{attribute 'linkalways'} 
{attribute 'no_explicit_call' := 'This FB is a CLASS and must be accessed using methods or properties'}
{attribute 'enable_dynamic_creation'}
FUNCTION_BLOCK Axis EXTENDS CyclicInstance
VAR
	_axisRef : Tc2_MC2.AXIS_REF;
	_power : MC_Power;
	_jog : MC_Jog;
	_readStatus : MC_ReadStatus;
	_parameterSet : ST_AxisParameterSet;
	
	_enable : BOOL;
	_enablePositive : BOOL;
	_enableNegative : BOOL;
	
	_override : LREAL := 100.0;
	_powerBufferMode : AxisBufferMode := AxisBufferMode.Aborting;
END_VAR

PROPERTY INTERNAL _InternalAxisRef : REFERENCE TO Tc2_MC2.AXIS_REF
GET
_InternalAxisRef REF= _axisRef;
END_GET
END_PROPERTY

PROPERTY INTERNAL _InternalJog : REFERENCE TO MC_Jog
GET
_InternalJog REF= _jog;
END_GET
END_PROPERTY

PROPERTY INTERNAL _InternalParameterSet : REFERENCE TO ST_AxisParameterSet
GET
_InternalParameterSet REF= _parameterSet;
END_GET
END_PROPERTY

PROPERTY AxisId : UDINT
GET
AxisId := _axisRef.NcToPlc.AxisId;
END_GET
END_PROPERTY

{warning 'add property implementation'}
PROPERTY BufferMode : Tc2_MC2.MC_BufferMode
GET
END_GET
SET
END_SET
END_PROPERTY

PROPERTY Busy : BOOL
GET
END_GET
END_PROPERTY

METHOD  CyclicCall
VAR_INST
	_readParameterSet : MC_ReadParameterSet;
	parameterSetRead : BOOL;
END_VAR
_power(
	Axis := THIS^._axisRef,
	Enable := THIS^._enable,
	Enable_Positive := THIS^._enablePositive,
	Enable_Negative := THIS^._enableNegative,
	Override := THIS^._override,
	BufferMode := THIS^._powerBufferMode
);

_readStatus(
	Axis := THIS^._axisRef,
	Enable := _enable
);

IF NOT parameterSetRead THEN
	_readParameterSet(
		Axis := THIS^._axisRef,
		Parameter := _parameterSet,
		Execute := TRUE
	);
	
	IF NOT _readParameterSet.Busy THEN
		_readParameterSet(
			Axis := THIS^._axisRef,
			Parameter := _parameterSet,
			Execute := TRUE
		);
		IF _readParameterSet.Done THEN
			parameterSetRead := TRUE;
		END_IF
	END_IF
END_IF
END_METHOD

METHOD Disable
_enable := FALSE;
END_METHOD

METHOD DisableNegative
_enableNegative := FALSE;
END_METHOD

METHOD DisablePositive
_enablePositive := FALSE;
END_METHOD

METHOD Enable
VAR_INPUT
	bufferMode : AxisBufferMode;
END_VAR
_enable := TRUE;
_powerBufferMode := bufferMode;
END_METHOD

METHOD EnableNegative : BOOL
_enableNegative := TRUE;
END_METHOD

METHOD EnablePositive
_enablePositive := TRUE;
END_METHOD

PROPERTY ErrorId : UDINT
GET
ErrorId := _readStatus.ErrorID;
END_GET
END_PROPERTY

METHOD Halt
VAR_INPUT
	feedback : REFERENCE TO I_CommandFeedback;
END_VAR
VAR_INST
	pCmd : POINTER TO HaltCommand;
END_VAR
pCmd := __NEW(HaltCommand(axisRef := THIS^));
pCmd^.Execute(feedback).ThenRelease();
END_METHOD

PROPERTY HasError : BOOL
GET
HasError := _readStatus.Error;
END_GET
END_PROPERTY

METHOD HomingBuilder : I_HomingBuilder
VAR_INST
	builder : DefaultHomingBuilder(axisRef := THIS^);
END_VAR
HomingBuilder := builder;
END_METHOD

PROPERTY IsAccelerating : BOOL
GET
IsAccelerating := _readStatus.Accelerating;
END_GET
END_PROPERTY

PROPERTY IsAtConstantVelocity : BOOL
GET
IsAtConstantVelocity := _readStatus.ConstantVelocity;
END_GET
END_PROPERTY

PROPERTY IsAtStandStill : BOOL
GET
IsAtStandStill := _readStatus.StandStill;
END_GET
END_PROPERTY

PROPERTY IsDecelerating : BOOL
GET
IsDecelerating := _readStatus.Decelerating;
END_GET
END_PROPERTY

PROPERTY IsErrorStopped : BOOL
GET
IsErrorStopped := _readStatus.ErrorStop;
END_GET
END_PROPERTY

PROPERTY IsHoming : BOOL
GET
IsHoming := _readStatus.Homing;
END_GET
END_PROPERTY

PROPERTY IsInContinuousMotion : BOOL
GET
IsInContinuousMotion := _readStatus.ContinuousMotion;
END_GET
END_PROPERTY

PROPERTY IsInDiscreteMotion : BOOL
GET
IsInDiscreteMotion := _readStatus.DiscreteMotion;
END_GET
END_PROPERTY

PROPERTY IsInSynchronizedMotion : BOOL
GET
IsInSynchronizedMotion := _readStatus.SynchronizedMotion;
END_GET
END_PROPERTY

PROPERTY IsReady : BOOL
GET
IsReady := _power.Status;
END_GET
END_PROPERTY

PROPERTY IsStatusValid : BOOL
GET
IsStatusValid := _readStatus.Valid;
END_GET
END_PROPERTY

PROPERTY IsStopping : BOOL
GET
IsStopping := _readStatus.Stopping;
END_GET
END_PROPERTY

METHOD JogBackwards
VAR_INPUT
	velocity : LREAL;
END_VAR
_jog(
	Axis := _axisRef,
	JogForward := FALSE,
	JogBackwards := TRUE,
	Mode := MC_JOGMODE_CONTINOUS,
	Velocity := velocity
);
END_METHOD

METHOD JogForward
VAR_INPUT
	velocity : LREAL;
END_VAR
_jog(
	Axis := _axisRef,
	JogForward := TRUE,
	JogBackwards := FALSE,
	Mode := MC_JOGMODE_CONTINOUS,
	Velocity := velocity
);
END_METHOD

METHOD MoveBuilder : I_MoveBuilder
VAR_INST
	builder : DefaultMoveBuilder(axisRef := THIS^);
END_VAR
MoveBuilder := builder;
END_METHOD

PROPERTY Override : LREAL
GET
Override := _override;
END_GET
SET
_override := Override;
END_SET
END_PROPERTY

METHOD Reset
VAR_INPUT
	feedback : REFERENCE TO I_CommandFeedback;
END_VAR
VAR_INST
	pCmd : POINTER TO ResetCommand;
END_VAR
pCmd := __NEW(ResetCommand(axisRef := THIS^));
pCmd^.Execute(feedback).ThenRelease();
END_METHOD

METHOD SetPositionAbsolute
VAR_INPUT
	positionToSet : LREAL;
	feedback : REFERENCE TO I_CommandFeedback;
END_VAR
VAR_INST
	pCmd : POINTER TO SetPositionCommand;
END_VAR
pCmd := __NEW(SetPositionCommand(axisRef := THIS^, position := positionToSet, mode := SetPositionMode.Absolute));
pCmd^.Execute(feedback).ThenRelease();
END_METHOD

METHOD SetPositionRelative
VAR_INPUT
	distanceToShift : LREAL;
	feedback : REFERENCE TO I_CommandFeedback;
END_VAR
VAR_INST
	pCmd : POINTER TO SetPositionCommand;
END_VAR
pCmd := __NEW(SetPositionCommand(axisRef := THIS^, position := distanceToShift, mode := SetPositionMode.Relative));
pCmd^.Execute(feedback).ThenRelease();
END_METHOD

METHOD Stop
VAR_INPUT
	feedback : REFERENCE TO I_CommandFeedback;
END_VAR
VAR_INST
	pCmd : POINTER TO StopCommand;
END_VAR
pCmd := __NEW(StopCommand(axisRef := THIS^));
pCmd^.Execute(feedback).ThenRelease();
END_METHOD

METHOD StopJogging
_jog(
	Axis := _axisRef,
	JogForward := FALSE,
	JogBackwards := FALSE,
);
END_METHOD

END_FUNCTION_BLOCK

(* stored: Version 1.1.0.1, ProductVersion 3.1.4024.12
   POU Axis: Id {2aaf2d97-dcbd-4e4f-bb30-8168c2228304}, SpecialFunc None
   Folder Actions: Id {d3a6f6e5-0dc6-41bb-8fed-2d69291737e9}
   Folder Builders: Id {8b93d50b-0153-46ae-83ea-c4e3e102f098}
   Folder Internal Methods: Id {a404c9ad-82b3-4270-92e5-46406a4ee946}
   Folder Internal Properties: Id {ff3545d4-cf9d-4f1c-9c6a-4608c8343033}
   Folder Properties: Id {bcfa7b74-d450-4ebb-b173-8da30bff7c11}
   Property _InternalAxisRef: Id {90609a99-e5bd-4b83-a58a-33c30ccc26cb}
   Get Get: Id {3b2ee038-497c-4033-a9b8-e83a2391191c}
   Property _InternalJog: Id {81758ae0-123d-466a-a4f8-f7ea636e9aab}
   Get Get: Id {8cd6a88b-f9db-4297-8b57-8b361f25d990}
   Property _InternalParameterSet: Id {247c45f2-47fd-4c00-8a9c-f77b32401e79}
   Get Get: Id {e12d2eff-e487-46f7-9fd3-f34e9951cc7f}
   Property AxisId: Id {67de2fd0-4aba-0578-2c2c-7b4e6a0d9ac8}
   Get Get: Id {821606fd-2277-088b-2511-fa15594f6c0e}
   Property BufferMode: Id {d3f9ce10-8ed2-4c86-bbbf-2cd31077c031}
   Get Get: Id {cb7a3b58-9630-4fcc-a8b2-6febff3711f9}
   Set Set: Id {90ad7435-fc63-4033-8f56-5ec9006dd1f3}
   Property Busy: Id {c365381d-4981-4e80-ad93-d15d1877f546}
   Get Get: Id {bb4c1cbb-227d-474b-b0fd-1dc32af91f9d}
   Method CyclicCall: Id {d18012b0-9520-4a5f-86ea-978a26c54f8e}
   Method Disable: Id {17b30872-fcd4-488a-b1b6-7fa79c000037}
   Method DisableNegative: Id {09f6abf1-b00f-4bfb-88e9-6ee7e9ba6e8f}
   Method DisablePositive: Id {59728fb8-b0dd-4aa9-bc80-abeb26875c9a}
   Method Enable: Id {c9911178-c912-485d-91e6-84927ecfc191}
   Method EnableNegative: Id {4800b13a-5042-4e28-861b-962c18550409}
   Method EnablePositive: Id {f7745032-8e58-4ba9-a609-48f560d8e17f}
   Property ErrorId: Id {ca7b6c5d-7148-4955-9c48-485f289f249e}
   Get Get: Id {248416d9-c77b-4a42-bcab-47b4bf745b98}
   Method Halt: Id {382b5bff-1007-4126-99ae-6487c254db90}
   Property HasError: Id {8b59e8d8-b8ff-463f-bd21-156952931aa9}
   Get Get: Id {ebd77229-528e-47c1-afbb-2dd2d9fa797c}
   Method HomingBuilder: Id {eff276be-bb3a-49d8-a728-ded3ab0a5295}
   Property IsAccelerating: Id {af076db1-4a05-447d-9648-e82349655e5d}
   Get Get: Id {3f9cd521-8eaf-450d-aeaa-ad5759d3a6ca}
   Property IsAtConstantVelocity: Id {a3739dbf-55c6-4ddc-b18a-6ca6e64d6d09}
   Get Get: Id {09f674dd-45ed-4115-a5f6-2d1775113eff}
   Property IsAtStandStill: Id {015a7b8b-a87e-4641-922b-b2dc302a276a}
   Get Get: Id {8da82d91-c4f0-439c-bd3d-90ccc4b5b090}
   Property IsDecelerating: Id {fee796ca-7d3a-4909-9ac5-028d4d20a128}
   Get Get: Id {c3ee7dee-9c69-4ca2-9379-dccd4ab16938}
   Property IsErrorStopped: Id {7db399a5-d190-443c-a64a-3aaf9b464e29}
   Get Get: Id {dcf2e2ef-7614-46d2-870d-814ff9464a9e}
   Property IsHoming: Id {1ddbd359-0a25-48b4-b010-3b06b077febf}
   Get Get: Id {4a60d080-4980-4525-b072-ea2241349744}
   Property IsInContinuousMotion: Id {d630d362-4c31-4edc-bbbc-0ee50039562c}
   Get Get: Id {44f97cb0-0fe0-4081-a420-5ac66cc2aee1}
   Property IsInDiscreteMotion: Id {55832b77-a03b-4968-80c6-15cdd3cedf1e}
   Get Get: Id {9ff7d675-0443-4b48-acce-a748fe5b301d}
   Property IsInSynchronizedMotion: Id {dcdf15cb-4b28-4e0e-9d50-c12a0ebeb79f}
   Get Get: Id {96ce6fd9-96bc-4849-aa22-4fe6df2c1bc4}
   Property IsReady: Id {b54c065f-5a64-4c0d-8d6f-34322fb086f7}
   Get Get: Id {35fca6b4-6504-482b-92aa-baa42de86f16}
   Property IsStatusValid: Id {5d176b49-ddfd-493b-a76c-4eedfca85975}
   Get Get: Id {3159d9ae-bc8b-4b0b-9615-6ab7905dbab0}
   Property IsStopping: Id {71248b21-bd4b-4d2b-8b0c-0bbaf737574b}
   Get Get: Id {a6e22c24-2be4-45bf-b856-bcb0459941d8}
   Method JogBackwards: Id {a7cfbd72-0a93-4039-b1d1-fcfceccd872a}
   Method JogForward: Id {cbd173e2-a265-46eb-94b8-308978a0bc52}
   Method MoveBuilder: Id {b4b2cd80-1567-4959-8de3-bde7b18dc77d}
   Property Override: Id {a8028f42-b9a9-4eb1-a0b7-86a2bf0543d0}
   Get Get: Id {5efb0fe9-a3fb-4d2d-9237-646a4db962e7}
   Set Set: Id {bb3b3dd2-c751-4d86-9a0c-4a3568e49fe6}
   Method Reset: Id {8e153cc3-92a5-4e6b-b7b2-9baa243ed4c1}
   Method SetPositionAbsolute: Id {889cfb23-a044-4223-ac9f-9539fa2ab6e4}
   Method SetPositionRelative: Id {b7781aa1-05ad-429c-b757-7906b6bcdcd3}
   Method Stop: Id {d6deae41-9d85-4fbd-8130-99bdb4cd48bd}
   Method StopJogging: Id {889afa4c-09c7-4dfc-8836-229afe5087d6} *)
